{attribute 'GeneratedUsingTerminal: EP3632-0001-0016'}
{attribute addProperty BoxType "EP3632-0001-0016"}
{attribute addProperty Id "STATUSAT %I*STATUS_B07533568"}
{attribute addProperty CRC "1971471493"}
{attribute addProperty Size "8"}
TYPE Ch2_Status_75824485 :
STRUCT
	{attribute addProperty Name "STATUS"}
	STATUS AT %I* : STATUS_B0753356;
END_STRUCT
END_TYPE

(* stored: Version 1.2.0.0, ProductVersion 3.1.4024.9
   DUT Ch2_Status_75824485: Id {aa2897fa-ca80-4b39-82b2-cdc925cec4cc} *)
